FUNCTION_BLOCK EHWCalculatePosition
VAR_INPUT
	rBarcodeReading : REAL; 	// current barcode reading
	tsTrack : Track_Segment;	// currentr track segment
END_VAR
VAR_OUTPUT
	rResult : REAL;
END_VAR
VAR
END_VAR

IF tsTrack.rStart < tsTrack.rEnd THEN
	rResult := tsTrack.rAbsoluteStart + (rBarcodeReading - tsTrack.rStart);
ELSE
	rResult := tsTrack.rAbsoluteEnd + (rBarcodeReading - tsTrack.rEnd);
END_IF

END_FUNCTION_BLOCK

(* stored: Version 1.1.0.1
   POU EHWCalculatePosition: Id {1693a63d-35b9-4247-862f-0fde8398dda6}, SpecialFunc None *)
